INTERFACE IEvent_ExecutionFailed EXTENDS IEvent

METHOD RaiseEx
VAR_INPUT
    Message : T_MaxString;
END_VAR
END_METHOD

END_INTERFACE

(* stored: Version 1.1.0.1, ProductVersion 3.1.4024.3
   Itf IEvent_ExecutionFailed: Id {8020b691-7dd5-07d7-319b-109e5a16216d}
   Method RaiseEx: Id {d168beec-4c21-0572-348b-075d7f983b25} *)
